FUNCTION_BLOCK FB_TestSuite2 EXTENDS FB_TestSuite
VAR_INPUT
END_VAR
VAR_OUTPUT
END_VAR
VAR
END_VAR

TestCase2A();
TestCase2B();

METHOD TestCase2A
VAR_INPUT
END_VAR
TEST('TestCase2A');

AssertTrue(TRUE, 'Condition is not true');

TEST_FINISHED();
END_METHOD

METHOD TestCase2B
VAR_INPUT
END_VAR
TEST('TestCase2B');

AssertTrue(TRUE, 'Condition is not true');
AssertTrue(TRUE, 'Condition is not true');

TEST_FINISHED();
END_METHOD

END_FUNCTION_BLOCK

(* stored: Version 1.1.0.1, ProductVersion 3.1.4024.12
   POU FB_TestSuite2: Id {3a6274d6-6083-4f38-89f5-174a468b61d8}, SpecialFunc None
   Method TestCase2A: Id {08302e5c-315f-491e-adf5-28ac987840cc}
   Method TestCase2B: Id {d124f6c2-5ec2-4271-8a1e-818da4d1bf79} *)
